FUNCTION_BLOCK IsMotorTick (* Basic Function Block Type *)
  (* Standard: 61499-2 *)
  (* Version 0.0, 21/06/2022, Lernfabrik, WBK hackaton, Template *)
  PACKAGE Main;
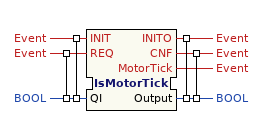
  EVENT_INPUT
    INIT WITH QI; (* Initialization Request *)
    REQ WITH QI; (* Normal Execution Request *)
  END_EVENT
  EVENT_OUTPUT
    INITO WITH Output; (* Initialization Confirm *)
    CNF WITH Output; (* Execution Confirmation *)
    MotorTick;
  END_EVENT
  VAR_INPUT
    QI : BOOL; (* Input event qualifier *)
  END_VAR
  VAR_OUTPUT
    Output : BOOL; (* Output event qualifier *)
  END_VAR
  VAR
    QS : BOOL;
  END_VAR
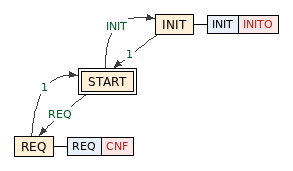
  EC_STATES
    START; (* Initial State *)
    INIT : INIT -> INITO; (* Initialization *)
    REQ : REQ -> CNF; (* Normal execution *)
  END_STATES
  EC_TRANSITIONS
    START TO INIT := INIT;
    INIT TO START := 1;
    START TO REQ := REQ;
    REQ TO START := 1;
  END_TRANSITIONS
  ALGORITHM INIT IN ST: (* Initialization algorithm *)
QS := 0;
  END_ALGORITHM
  ALGORITHM REQ IN ST: (* Normally executed algorithm *)
(* Bei jedem Motorschritt ( = Change im Motorwert ) wird ein Output gegeben *)
IF QI = QS THEN
	Output := 1;
	MotorTick := 1;
END_IF;

QS := NOT QI;
  END_ALGORITHM
END_FUNCTION_BLOCK
